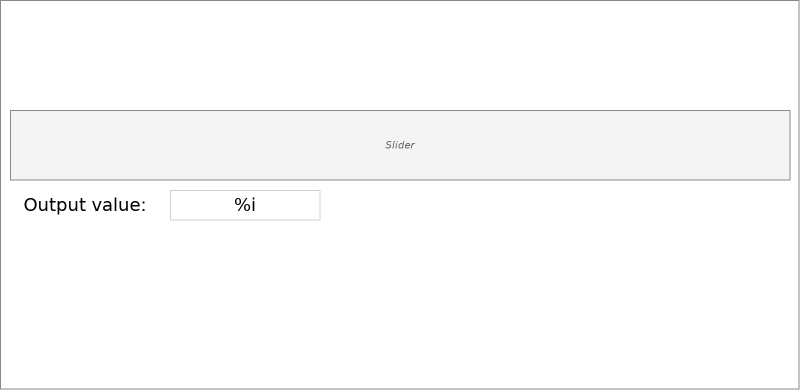
VISUALIZATION VisuAnalogOutControl  // 800x390
    Slider (10,110 780x70), variable: GVL_DevManual.fbManualControler.pDevAnalogOut^.fCmdValue, scale 0..100
    Textfield (170,190 150x30), "%i", text variable: GVL_DevManual.fbManualControler.pDevAnalogOut^.fCmdValue
        OnMouseClick: write the text variable via VisuDialogs.Numpad
    Label (10,190 150x30), "Output value:"
END_VISUALIZATION

(* stored: Version 1.1.0.1, ProductVersion 3.1.4024.5
   Visu VisuAnalogOutControl: Id {6054b02d-98e9-4d8c-9154-935e2b6b306b} *)
